FUNCTION_BLOCK Switchtank
  (* Standard: 61499-2 *)
  (* Version 0,1, 2015-00-10, Th?o, PC_THEO *)
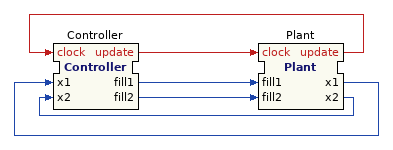
  FBS
    Controller : Controller;
    Plant : Plant;
  END_FBS
  EVENT_CONNECTIONS
    Controller.update TO Plant.clock;
    Plant.update TO Controller.clock;
  END_CONNECTIONS
  DATA_CONNECTIONS
    Controller.fill1 TO Plant.fill1;
    Controller.fill2 TO Plant.fill2;
    Plant.x1 TO Controller.x1;
    Plant.x2 TO Controller.x2;
  END_CONNECTIONS
END_FUNCTION_BLOCK
